{attribute 'linkalways'} 
{attribute 'no_explicit_call' := 'This FB is a CLASS and must be accessed using methods or properties'}
{attribute 'enable_dynamic_creation'}
FUNCTION_BLOCK Node_F_VN_ReferenceColorSimilarity_TcVnVector3_LREAL EXTENDS VisionNode
VAR
	ipSrcImage : _ITcVnImage;
    ipDestImage : _ITcVnImage;
    aRefColor : _TcVnVector3_LREAL;
    hrPrev : _HRESULT(S_OK);
	hresult : _HRESULT(S_OK);
END_VAR

METHOD PUBLIC  Clone : I_Node
VAR
	pNode : POINTER TO Node_F_VN_ReferenceColorSimilarity_TcVnVector3_LREAL;
END_VAR
pNode := __NEW(Node_F_VN_ReferenceColorSimilarity_TcVnVector3_LREAL);
Clone := pNode^;
END_METHOD

METHOD FB_init : BOOL
VAR_INPUT
	bInitRetains : BOOL; // if TRUE, the retain variables are initialized (warm start / cold start)
	bInCopyCode : BOOL;  // if TRUE, the instance afterwards gets moved into the copy code (online change)
END_VAR
AddInput('ipSrcImage', ipSrcImage);
AddInput('aRefColor', aRefColor);
AddInput('hrPrev', hrPrev);
AddOutput('ipDestImage', ipDestImage);
AddOutput('hresult', hresult);
END_METHOD

METHOD PROTECTED OnExecute
hresult.Value := F_VN_ReferenceColorSimilarity_TcVnVector3_LREAL(
	ipSrcImage := ipSrcImage.Value,
    ipDestImage := ipDestImage.Value,
    aRefColor := aRefColor.Value,
	hrPrev := hrPrev.Value);
END_METHOD

METHOD PUBLIC PreExecutionCheck
VAR_INPUT
	Check : I_PreExecutionChecks;
END_VAR
VAR
    colorMapSize : ULINT;
END_VAR
Check.IsTrue(ipSrcImage.IsValid, 'ipSrcImage must contain an image');
Check.IsTrue(ipSrcImage.HasChannelCount(3), 'ipSrcImage must have 3 channels');
Check.IsTrue(ipSrcImage.IsPixelDepth(8), 'ipSrcImage must have 8 bit pixel depth');
END_METHOD

END_FUNCTION_BLOCK

(* stored: Version 1.1.0.1, ProductVersion 3.1.4024.15
   POU Node_F_VN_ReferenceColorSimilarity_TcVnVector3_LREAL: Id {f581cc75-5379-0dd6-391e-7cbdbd9e1327}, SpecialFunc None
   Folder Constructor: Id {d8fcf3af-31cf-021b-0be9-a9a1051f6047}
   Method Clone: Id {783e86a3-ae8e-05cf-392f-2eba18ad5c32}
   Method FB_init: Id {27e1433e-efbf-09c5-0122-6c022dcaa260}
   Method OnExecute: Id {c496a791-7776-09b9-2376-16bb92a38636}
   Method PreExecutionCheck: Id {555533cd-e2bf-0349-28d3-344d889e66c1} *)
